// TIA Portal project "Conveyor and Puncher" (V17)
// Conveyor Line with Rejection
// The conveyor should stop for 10 seconds and a puncher will be ON for 2 seconds, when a defect is detected.

(* hardware
DEVICE "S7-1200 station_1"  S7-1200 Station
   slot 0: "Rack_0"  S7-1200 Rack  Rack  V1.0
   slot 1: "PLC_1"  CPU 1212C DC/DC/DC  6ES7 212-1AE40-0XB0  V4.5
*)

// ===== PLC "PLC_1"  CPU 1212C DC/DC/DC =====

VAR_GLOBAL   // PLC tag table "Default tag table"
   "PB" AT %I0.0 : Bool;
   "Vision_Sensor" AT %I0.1 : Bool;
   "Conveyor" AT %Q0.0 : Bool;
   "Puncher" AT %Q0.1 : Bool;
   "Tag_1" AT %M0.0 : Bool;
   "Tag_2" AT %M0.1 : Bool;
END_VAR

// folder: System blocks/Program resources

DATA_BLOCK "IEC_Timer_0_DB"   // DB1
{ S7_Optimized_Access := 'TRUE' }
AUTHOR : Simatic
FAMILY : IEC
NAME : IEC_TMR
VERSION : 1.0
// stored: InstanceOfName IEC_TIMER
"IEC_TIMER"
BEGIN
END_DATA_BLOCK

DATA_BLOCK "IEC_Timer_0_DB_1"   // DB2
{ S7_Optimized_Access := 'TRUE' }
AUTHOR : Simatic
FAMILY : IEC
NAME : IEC_TMR
VERSION : 1.0
// stored: InstanceOfName IEC_TIMER
"IEC_TIMER"
BEGIN
END_DATA_BLOCK

// folder: (top level)

ORGANIZATION_BLOCK "Main"   // OB1, LAD, ProgramCycle
TITLE = "Main Program Sweep (Cycle)"
{ S7_Optimized_Access := 'TRUE' }
VERSION : 0.1
   VAR_INPUT
      Initial_Call : Bool;   // Initial call of this OB
      Remanence : Bool;   // =True, if remanent data are available
   END_VAR
BEGIN

REGION Network 1
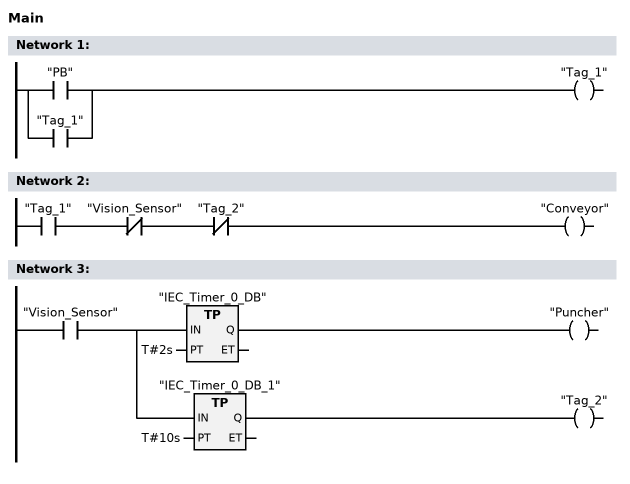
   RUNG wire#powerrail
      Contact( "PB" )
      wire#w1
      Coil( "Tag_1" )
   END_RUNG
   RUNG wire#powerrail
      Contact( "Tag_1" )
   END_RUNG wire#w1
   // the same network as SCL:
   "Tag_1" := "PB" OR "Tag_1";
END_REGION

REGION Network 2
   RUNG wire#powerrail
      Contact( "Tag_1" )
      I_Contact( "Vision_Sensor" )
      I_Contact( "Tag_2" )
      Coil( "Conveyor" )
   END_RUNG
   // the same network as SCL:
   "Conveyor" := "Tag_1" AND NOT "Vision_Sensor" AND NOT "Tag_2";
END_REGION

REGION Network 3
   "IEC_Timer_0_DB".TP(IN := "Vision_Sensor", PT := T#2s);
   "Puncher" := "IEC_Timer_0_DB".Q;
   "IEC_Timer_0_DB_1".TP(IN := "Vision_Sensor", PT := T#10s);
   "Tag_2" := "IEC_Timer_0_DB_1".Q;
END_REGION
END_ORGANIZATION_BLOCK